INTERFACE I_MessageData

PROPERTY DirRoot : POINTER to string(255)
SET
END_SET
END_PROPERTY

PROPERTY ErrorIndex : reference to uint
SET
END_SET
END_PROPERTY

PROPERTY FileRoot : pointer to string(255)
SET
END_SET
END_PROPERTY

PROPERTY LocalTime : pointer to DT
SET
END_SET
END_PROPERTY

PROPERTY MessageIndex : reference to uint
SET
END_SET
END_PROPERTY

PROPERTY MsgList : pointer to ARRAY[1..GVL_MSG_XTS.MAX_MESSAGE] OF st_message
SET
END_SET
END_PROPERTY

END_INTERFACE

(* stored: Version 1.1.0.1, ProductVersion 3.1.4026.18
   Itf I_MessageData: Id {2db9b6a6-428d-4711-b7d7-1c3cb7282175}
   Property DirRoot: Id {7a7660f6-8dd0-4241-8cdf-d9a8471bf5da}
   Set Set: Id {fc7b1e2c-2722-4569-ad96-6e083b12db94}
   Property ErrorIndex: Id {ca44583b-b425-476e-a5cd-c6caf82fddd4}
   Set Set: Id {360c4630-de54-4e72-badc-523252289b1e}
   Property FileRoot: Id {93a7f7ac-a718-4a99-bedf-784f478e8139}
   Set Set: Id {d51caa8b-cda6-4e15-90b5-1f3b095e2d34}
   Property LocalTime: Id {4a8c6cf9-bb8f-4430-90ec-72c237df6821}
   Set Set: Id {59454843-3397-4267-94b3-a2f46589d066}
   Property MessageIndex: Id {72b1ed0c-73fa-4f83-bf7d-cdb62d320b0c}
   Set Set: Id {a121c52d-964c-49e6-96ee-8c1438957c98}
   Property MsgList: Id {bb7a9b1f-c91a-4135-9e66-93d6c1f1c5d5}
   Set Set: Id {bc0efa70-3e08-4c72-8462-c70d3560f13c} *)
